{attribute addProperty BoxType "EJ1918-0000-0017"}
{attribute addProperty Id "FSoE_InputsFSoE_Inputs_2B542CE7567FSoE_OutputsFSoE_Outputs_F12FD39F486"}
{attribute addProperty CRC "2580529326"}
{attribute addProperty SizeInBites "104"}
{attribute addProperty SizeInBytes "13"}
TYPE Module_1_FSOE_99CFC0AE :
STRUCT
	{attribute addProperty Name "FSoE_Inputs"}
	FSoE_Inputs  : FSoE_Inputs_2B542CE7;
	{attribute addProperty Name "FSoE_Outputs"}
	FSoE_Outputs  : FSoE_Outputs_F12FD39F;
END_STRUCT
END_TYPE

(* stored: Version 1.2.0.0, ProductVersion 3.1.4024.9
   DUT Module_1_FSOE_99CFC0AE: Id {7ed472a4-58f3-4a91-9c23-fb16c1f6a95e} *)
